{attribute 'GeneratedUsingTerminal: KL6551'}
{attribute addProperty BoxType "KL6551"}
{attribute addProperty Id "Channel_1AT %Q*Channel_6931CC5B0"}
{attribute addProperty CRC "1384833944"}
{attribute addProperty Size "0"}
TYPE KL6551_528AE398 :
STRUCT
	{attribute addProperty Name "Channel_1"}
	Channel_1 : Channel_6931CC5B;
END_STRUCT
END_TYPE
